// Interlock logic for the Dump Chiller
FUNCTION F_DumpChillerEnable : BOOL
VAR_INPUT
    //bMasterOverride : BOOL; //Master manual override control input
    Mode : E_Mode;
END_VAR
VAR_IN_OUT CONSTANT
    stErrors : ST_ErrorStates; // Currently detected errors
END_VAR
VAR
END_VAR

IF (stErrors.bHardwareFailure // Disable dump chiller if there's a hardware failure
    //OR stErrors.bLeakOpticalTableAmphosOn OR stErrors.bLeakOpticalTableNoLaser OR stErrors.bLeakOpcpaCarbideOn OR stErrors.bLeakUnderTable) // Disable dump chiller for these leak conditions
   OR stErrors.bLeakUnderTable) 
   OR ( NOT (MODE = E_Mode.MASTER_Override))
THEN
    F_DumpChillerEnable := FALSE;
ELSE
	F_DumpChillerEnable := TRUE;
END_IF

END_FUNCTION

(* stored: Version 1.1.0.1, ProductVersion 3.1.4024.12
   POU F_DumpChillerEnable: Id {eacb95fa-49ef-4c8d-8057-f0d541675cea}, SpecialFunc None *)
